// SIMATIC STEP 7 (V5.x) project ZEn01_10_STEP7__Com_SFB
// CPU: CPU414-1(1)
// CPU: CPU416-1(1)
// station: Hardware
// station: SIMATIC 400-RCV
// station: Hardware
// station: SIMATIC 400-SEND
// program: S7 Receive-Program
// program: S7 Send-Program

SYMBOL_TABLE
"IDB_USEND"	DB 8	SFB 8
"IDB_URCV"	DB 9	SFB 9
"IDB_BSEND"	DB 12	SFB 12
"IDB_BRCV"	DB 13	SFB 13
"IDB_GET"	DB 14	SFB 14
"IDB_PUT"	DB 15	SFB 15
"IDB_START"	DB 19	SFB 19
"IDB_STOP"	DB 20	SFB 20
"IDB_RESUME"	DB 21	SFB 21
"IDB_STATUS"	DB 22	SFB 22
"IDB_USTATUS"	DB 23	SFB 23
"data_usend"	DB 100	DB 100
"data_urcv"	DB 101	DB 101
"data_bsend"	DB 102	DB 102
"data_brcv"	DB 103	DB 103
"data_get"	DB 104	DB 104
"data_put"	DB 105	DB 105
"data_program_cntr"	DB 106	DB 106	// Parameters SFB START , STOP,  RESUME, STATUS and USTATUS
"data_get_source"	DB 107	DB 107
"data_put_destination"	DB 108	DB 108
"CHECK"	FC 99	FC 99	// Check the control parameters of communication function blocks
"EXAMPLE_USEND"	FC 100	FC 100
"EXAMPLE_PUT"	FC 101	FC 101
"EXAMPLE_STOP"	FC 102	FC 102
"EXAMPLE_STATUS"	FC 103	FC 103
"EXAMPLE_URCV"	FC 104	FC 104
"EXAMPLE_BSEND"	FC 105	FC 105
"EXAMPLE_BRCV"	FC 106	FC 106
"EXAMPLE_GET"	FC 107	FC 107
"EXAMPLE_START"	FC 108	FC 108
"EXAMPLE_RESUME"	FC 109	FC 109
"EXAMPLE_USTATUS"	FC 110	FC 110
"EXAMPLE_PRESET_SFBs_1"	FC 111	FC 111	// Presets on Send-CPU
"EXAMPLE_PRESET_SFBs_2"	FC 112	FC 112	// Presets on Rcv-CPU
"req_usend_user"	M 20.0	BOOL	// Trigger USEND    0->1
"req_bsend_user"	M 20.2	BOOL	// Trigger BSEND    0->1
"req_get_user"	M 20.4	BOOL	// Trigger GET    0->1
"req_put_user"	M 20.5	BOOL	// Trigger PUT   0->1
"req_start_user"	M 20.6	BOOL	// Trigger START    0->1
"req_stop_user"	M 20.7	BOOL	// Trigger STOP    0->1
"req_resume_user"	M 21.0	BOOL	// Trigger RESUME    0->1
"req_status_user"	M 21.1	BOOL	// Trigger STATUS    0->1
"req_ustatus_user"	M 21.2	BOOL	// Trigger USTATUS    0->1
"CYCL_EXC"	OB 1	OB 1	// Cycle Execution
"CYC_INT5"	OB 35	OB 35	// Cyclic Interrupt 5
"COMPLETE RESTART"	OB 100	OB 100	// Complete Restart
"USEND"	SFB 8	SFB 8	// Uncoordinated Send
"URCV"	SFB 9	SFB 9	// Uncoordinated Receive
"BSEND"	SFB 12	SFB 12	// Block Oriented Send
"BRCV"	SFB 13	SFB 13	// Block Oriented Receive
"GET"	SFB 14	SFB 14	// Read Data From a Remote CPU
"PUT"	SFB 15	SFB 15	// Write Data to a Remote CPU
"START"	SFB 19	SFB 19	// Remote Start
"STOP"	SFB 20	SFB 20	// Remote Stop
"RESUME"	SFB 21	SFB 21	// Remote Restart
"STATUS"	SFB 22	SFB 22	// Remote Status
"USTATUS"	SFB 23	SFB 23	// Receive Remote Status
"FILL"	SFC 21	SFC 21
END_SYMBOL_TABLE

FUNCTION "CHECK" : VOID	// FC 99
//This block is used to evaluate the parameters DONE/NDR/ERROR/STATUS for the 
//CFBs. 
//The parameters OK/NOT_OK are set depending on the passed parameters. 
//
VERSION : 0.0
VAR_INPUT
  ERROR : BOOL ;
  STATUS : WORD ;
  DONE_NDR : BOOL ;
END_VAR
VAR_OUTPUT
  OK : BOOL ;	// 0 Error/warning while executing CFB
  NOT_OK : BOOL ;
END_VAR
VAR_TEMP
  STAT : BOOL ;
END_VAR
BEGIN
NETWORK
TITLE = This block can be used for troubleshooting if needed
      L     #STATUS;	// Check STATUS
      L     0;
      <>I;
      =     #STAT;	// Error/warning while executing CFB 
      A     #DONE_NDR;
      =     #OK;	// CFB execution OK
      O     #STAT;	// WARNING/ERROR
      O     #ERROR;	// ERROR
      R     #OK;	// CFB execution not OK
      S     #NOT_OK;
END_FUNCTION

FUNCTION "EXAMPLE_USEND" : VOID	// FC 100
//Controlling USEND 
//
VERSION : 2.0
BEGIN
NETWORK
TITLE =
      A     "req_usend_user";	//*If "req" 0->1,
      JCN   m1;
      L     0;	//*reset 
      T     "data_usend".saved_status;	//*saved STATUS 
m1:   NOP   0;
      BLD   9;
      =     L 4.0;
      CDB;
      OPN   DI 8;
      TAR2  LD 0;
      A     "req_usend_user";
      =     DIX 0.0;
      OPN   DI 100;
      L     DIW 2;
      OPN   DI 8;
      T     DIW 2;
      OPN   DI 100;	//*If STATUS is not "0",
      L     DID 4;	//*
      OPN   DI 8;	//*
      T     DID 4;
      L     W#16#1002;	//*
      T     DIW 12;	//*set "not_ok"
      L     30;	//*and save STATUS
      T     DIW 14;
      L     100;	//*If "done"
      T     DIW 16;	//*or "error"
      L     P#DBX 10.0;	//*reset "req"
      T     DID 18;
//                                      //Add troubleshooting routine here
      L     W#16#1002;
      T     DIW 22;
      L     30;
      T     DIW 24;
      L     100;
      T     DIW 26;
      L     P#DBX 110.0;
      T     DID 28;
      L     W#16#1002;
      T     DIW 32;
      L     30;
      T     DIW 34;
      L     100;
      T     DIW 36;
      L     P#DBX 210.0;
      T     DID 38;
      L     W#16#1002;
      T     DIW 42;
      L     30;
      T     DIW 44;
      L     100;
      T     DIW 46;
      L     P#DBX 310.0;
      T     DID 48;
      LAR2  P#DBX 0.0;
      UC    "USEND";
      LAR2  LD 0;
      A     DIX 8.0;
      OPN   DI 100;
      =     DIX 0.1;
      OPN   DI 8;
      A     DIX 8.1;
      OPN   DI 100;
      =     DIX 0.2;
      OPN   DI 8;
      L     DIW 10;
      OPN   DI 100;
      T     DIW 8;
      OPN   DI 8;
      CDB;
      BLD   10;
      L     0;
      L     "data_usend".status;
      <>I;
      JCN   mark;
      SET;
      =     "data_usend".not_ok;
      T     "data_usend".saved_status;
mark: NOP   0;
      A     "data_usend".done;
      O     "data_usend".error;
      R     "req_usend_user";
      A     "data_usend".not_ok;
END_FUNCTION

FUNCTION "EXAMPLE_PUT" : VOID	// FC 101
VERSION : 2.0
BEGIN
NETWORK
TITLE =
      A     "req_put_user";	//*If "req" 0->1,
      JCN   m1;
      L     0;	//*reset 
      T     "data_put".saved_status;	//*saved STATUS 
m1:   NOP   0;
      BLD   9;
      =     L 4.0;
      CDB;
      OPN   DI 15;
      TAR2  LD 0;
      A     "req_put_user";
      =     DIX 0.0;
      OPN   DI 105;
      L     DIW 2;
      OPN   DI 15;
      T     DIW 2;
      L     W#16#1002;
      T     DIW 8;
      L     100;
      T     DIW 10;	//*If STATUS is not "0",
      L     108;	//*
      T     DIW 12;	//*
      L     P#DBX 0.0;
      T     DID 14;	//*
      L     W#16#1002;	//*set "not_ok"
      T     DIW 18;	//*and save STATUS
      L     100;
      T     DIW 20;	//*If "done"
      L     108;	//*or "error"
      T     DIW 22;	//*reset "req"
      L     P#DBX 100.0;
//                                      //Add troubleshooting routine here
      T     DID 24;
      L     W#16#1002;
      T     DIW 28;
      L     100;
      T     DIW 30;
      L     108;
      T     DIW 32;
      L     P#DBX 200.0;
      T     DID 34;
      L     W#16#1002;
      T     DIW 38;
      L     100;
      T     DIW 40;
      L     108;
      T     DIW 42;
      L     P#DBX 300.0;
      T     DID 44;
      L     W#16#1002;
      T     DIW 48;
      L     100;
      T     DIW 50;
      L     105;
      T     DIW 52;
      L     P#DBX 6.0;
      T     DID 54;
      L     W#16#1002;
      T     DIW 58;
      L     100;
      T     DIW 60;
      L     105;
      T     DIW 62;
      L     P#DBX 106.0;
      T     DID 64;
      L     W#16#1002;
      T     DIW 68;
      L     100;
      T     DIW 70;
      L     105;
      T     DIW 72;
      L     P#DBX 206.0;
      T     DID 74;
      L     W#16#1002;
      T     DIW 78;
      L     100;
      T     DIW 80;
      L     105;
      T     DIW 82;
      L     P#DBX 306.0;
      T     DID 84;
      LAR2  P#DBX 0.0;
      UC    "PUT";
      LAR2  LD 0;
      A     DIX 4.0;
      OPN   DI 105;
      =     DIX 0.1;
      OPN   DI 15;
      A     DIX 4.1;
      OPN   DI 105;
      =     DIX 0.2;
      OPN   DI 15;
      L     DIW 6;
      OPN   DI 105;
      T     DIW 4;
      OPN   DI 15;
      CDB;
      BLD   10;
      L     0;
      L     "data_put".status;
      <>I;
      JCN   mark;
      SET;
      =     "data_put".not_ok;
      T     "data_put".saved_status;
mark: NOP   0;
      A     "data_put".done;
      O     "data_put".error;
      R     "req_put_user";
      A     "data_put".not_ok;
END_FUNCTION

FUNCTION "EXAMPLE_STOP" : VOID	// FC 102
VERSION : 2.0
BEGIN
NETWORK
TITLE =
      A     "req_stop_user";	//*If "req" 0->1,
      JCN   m1;
      L     0;	//*reset 
      T     "data_program_cntr".stp_saved_status;	//*saved STATUS 
m1:   NOP   0;
      BLD   9;
      =     L 4.0;
      CDB;
      OPN   DI 20;
      TAR2  LD 0;
      A     "req_stop_user";
      =     DIX 0.0;
      OPN   DI 106;
      L     DIW 18;	//*If STATUS is not "0",
      OPN   DI 20;	//*
      T     DIW 2;	//*
      L     W#16#1002;
      T     DIW 8;	//*
      L     10;	//*set "not_ok"
      T     DIW 10;	//*and save STATUS
      L     106;
      T     DIW 12;	//*If "done"
      L     P#DBX 0.0;	//*or "error"
      T     DID 14;	//*reset "req"
      OPN   DI 106;	//                                      //Add troubleshooting routine here
      L     DIB 22;
      OPN   DI 20;
      T     DIB 18;
      LAR2  P#DBX 0.0;
      UC    "STOP";
      LAR2  LD 0;
      A     DIX 4.0;
      OPN   DI 106;
      =     DIX 17.1;
      OPN   DI 20;
      A     DIX 4.1;
      OPN   DI 106;
      =     DIX 17.2;
      OPN   DI 20;
      L     DIW 6;
      OPN   DI 106;
      T     DIW 20;
      OPN   DI 20;
      L     DIB 18;
      OPN   DI 106;
      T     DIB 22;
      OPN   DI 20;
      CDB;
      BLD   10;
      L     0;
      L     "data_program_cntr".stop_status;
      <>I;
      JCN   mark;
      SET;
      =     "data_program_cntr".stop_not_ok;
      T     "data_program_cntr".stp_saved_status;
mark: NOP   0;
      A     "data_program_cntr".stop_done;
      O     "data_program_cntr".stop_error;
      R     "req_stop_user";
      A     "data_program_cntr".stop_not_ok;
END_FUNCTION

FUNCTION "EXAMPLE_STATUS" : VOID	// FC 103
VERSION : 2.0
BEGIN
NETWORK
TITLE =
      A     "req_status_user";	//*If "req" 0->1,
      JCN   m1;
      L     0;	//*reset 
      T     "data_program_cntr".sta_saved_status;	//*saved STATUS 
m1:   NOP   0;
      BLD   9;
      =     L 4.0;
      CDB;
      OPN   DI 22;
      TAR2  LD 0;
      A     "req_status_user";
      =     DIX 0.0;
      OPN   DI 106;
      L     DIW 30;
      OPN   DI 22;	//*If STATUS is not "0",
      T     DIW 2;	//*
      L     W#16#1004;	//*
      T     DIW 8;
      L     1;	//*
      T     DIW 10;	//*set "not_ok"
      L     106;	//*and save STATUS
      T     DIW 12;
      L     P#DBX 34.0;	//*If "done"
      T     DID 14;	//*or "error"
      L     W#16#1004;	//*reset "req"
      T     DIW 18;
//                                      //Add troubleshooting routine here
      L     1;
      T     DIW 20;
      L     106;
      T     DIW 22;
      L     P#DBX 36.0;
      T     DID 24;
      L     W#16#1004;
      T     DIW 28;
      L     1;
      T     DIW 30;
      L     106;
      T     DIW 32;
      L     P#DBX 38.0;
      T     DID 34;
      LAR2  P#DBX 0.0;
      UC    "STATUS";
      LAR2  LD 0;
      A     DIX 4.0;
      OPN   DI 106;
      =     DIX 29.1;
      OPN   DI 22;
      A     DIX 4.1;
      OPN   DI 106;
      =     DIX 29.2;
      OPN   DI 22;
      L     DIW 6;
      OPN   DI 106;
      T     DIW 32;
      OPN   DI 22;
      CDB;
      BLD   10;
      L     0;
      L     "data_program_cntr".status_status;
      <>I;
      JCN   mark;
      SET;
      =     "data_program_cntr".status_not_ok;
      T     "data_program_cntr".sta_saved_status;
mark: NOP   0;
      A     "data_program_cntr".status_done;
      O     "data_program_cntr".status_error;
      R     "req_status_user";
      A     "data_program_cntr".status_not_ok;
END_FUNCTION

FUNCTION "EXAMPLE_BSEND" : VOID	// FC 105
//Controlling BSEND 
//
VERSION : 2.0
BEGIN
NETWORK
TITLE =
      A     "req_bsend_user";	//*If "req" 0->1,
      JCN   m1;
      L     0;	//*reset 
      T     "data_bsend".saved_status;	//*saved STATUS 
m1:   NOP   0;
      BLD   9;
      =     L 4.0;
      CDB;
      OPN   DI 12;
      TAR2  LD 0;
      A     "req_bsend_user";
      =     DIX 0.0;
      OPN   DI 102;
      L     DIW 2;
      OPN   DI 12;
      T     DIW 2;	//*If STATUS is not "0",
      OPN   DI 102;	//*
      L     DID 4;	//*
      OPN   DI 12;
      T     DID 4;	//*
      L     W#16#1002;	//*set "not_ok"
      T     DIW 12;	//*and save STATUS
      L     500;
      T     DIW 14;	//*If "done"
      L     102;	//*or "error"
      T     DIW 16;	//*reset "req"
      L     P#DBX 12.0;
//                                      //Add troubleshooting routine here
      T     DID 18;
      OPN   DI 102;
      L     DIW 10;
      OPN   DI 12;
      T     DIW 22;
      LAR2  P#DBX 0.0;
      UC    "BSEND";
      LAR2  LD 0;
      A     DIX 8.0;
      OPN   DI 102;
      =     DIX 0.1;
      OPN   DI 12;
      A     DIX 8.1;
      OPN   DI 102;
      =     DIX 0.2;
      OPN   DI 12;
      L     DIW 10;
      OPN   DI 102;
      T     DIW 8;
      OPN   DI 12;
      L     DIW 22;
      OPN   DI 102;
      T     DIW 10;
      OPN   DI 12;
      CDB;
      BLD   10;
      L     0;
      L     "data_bsend".status;
      <>I;
      JCN   mark;
      SET;
      =     "data_bsend".not_ok;
      T     "data_bsend".saved_status;
mark: NOP   0;
      A     "data_bsend".done;
      O     "data_bsend".error;
      R     "req_bsend_user";
      A     "data_bsend".not_ok;
END_FUNCTION

FUNCTION "EXAMPLE_GET" : VOID	// FC 107
VERSION : 2.0
BEGIN
NETWORK
TITLE =
      A     "req_get_user";	//*If "req" 0->1,
      JCN   m1;
      L     0;	//*reset 
      T     "data_get".saved_status;	//*saved STATUS 
m1:   NOP   0;
      BLD   9;
      =     L 4.0;
      CDB;
      OPN   DI 14;
      TAR2  LD 0;
      A     "req_get_user";
      =     DIX 0.0;
      OPN   DI 104;
      L     DIW 2;
      OPN   DI 14;
      T     DIW 2;
      L     W#16#1002;
      T     DIW 8;
      L     100;
      T     DIW 10;	//*If STATUS is not "0",
      L     107;	//*
      T     DIW 12;	//*
      L     P#DBX 0.0;
      T     DID 14;	//*
      L     W#16#1002;	//*set "not_ok"
      T     DIW 18;	//*and save STATUS
      L     100;
      T     DIW 20;	//*If "done"
      L     107;	//*or "error"
      T     DIW 22;	//*reset "req"
      L     P#DBX 100.0;
//                                      //Add troubleshooting routine here
      T     DID 24;
      L     W#16#1002;
      T     DIW 28;
      L     100;
      T     DIW 30;
      L     107;
      T     DIW 32;
      L     P#DBX 200.0;
      T     DID 34;
      L     W#16#1002;
      T     DIW 38;
      L     100;
      T     DIW 40;
      L     107;
      T     DIW 42;
      L     P#DBX 300.0;
      T     DID 44;
      L     W#16#1002;
      T     DIW 48;
      L     100;
      T     DIW 50;
      L     104;
      T     DIW 52;
      L     P#DBX 6.0;
      T     DID 54;
      L     W#16#1002;
      T     DIW 58;
      L     100;
      T     DIW 60;
      L     104;
      T     DIW 62;
      L     P#DBX 106.0;
      T     DID 64;
      L     W#16#1002;
      T     DIW 68;
      L     100;
      T     DIW 70;
      L     104;
      T     DIW 72;
      L     P#DBX 206.0;
      T     DID 74;
      L     W#16#1002;
      T     DIW 78;
      L     100;
      T     DIW 80;
      L     104;
      T     DIW 82;
      L     P#DBX 306.0;
      T     DID 84;
      LAR2  P#DBX 0.0;
      UC    "GET";
      LAR2  LD 0;
      A     DIX 4.0;
      OPN   DI 104;
      =     DIX 0.1;
      OPN   DI 14;
      A     DIX 4.1;
      OPN   DI 104;
      =     DIX 0.2;
      OPN   DI 14;
      L     DIW 6;
      OPN   DI 104;
      T     DIW 4;
      OPN   DI 14;
      CDB;
      BLD   10;
      L     0;
      L     "data_get".status;
      <>I;
      JCN   mark;
      SET;
      =     "data_get".not_ok;
      T     "data_get".saved_status;
mark: NOP   0;
      A     "data_get".ndr;
      O     "data_get".error;
      R     "req_get_user";
      A     "data_get".not_ok;
END_FUNCTION

FUNCTION "EXAMPLE_START" : VOID	// FC 108
VERSION : 2.0
BEGIN
NETWORK
TITLE =
      A     "req_start_user";	//*If "req" 0->1,
      JCN   m1;
      L     0;	//*reset 
      T     "data_program_cntr".stt_saved_status;	//*saved STATUS 
m1:   NOP   0;
      BLD   9;
      =     L 4.0;
      CDB;
      OPN   DI 19;
      TAR2  LD 0;
      A     "req_start_user";
      =     DIX 0.0;
      OPN   DI 106;
      L     DIW 12;
      OPN   DI 19;	//*If STATUS is not "0",
      T     DIW 2;	//*
      L     W#16#1002;	//*
      T     DIW 8;
      L     10;	//*
      T     DIW 10;	//*set "not_ok"
      L     106;	//*and save STATUS
      T     DIW 12;
      L     P#DBX 0.0;	//*If "done"
      T     DID 14;	//*or "error"
      OPN   DI 106;	//*reset "req"
      L     DIB 16;
//                                      //Add troubleshooting routine here
      OPN   DI 19;
      T     DIB 28;
      LAR2  P#DBX 0.0;
      UC    "START";
      LAR2  LD 0;
      A     DIX 4.0;
      OPN   DI 106;
      =     DIX 10.1;
      OPN   DI 19;
      A     DIX 4.1;
      OPN   DI 106;
      =     DIX 10.2;
      OPN   DI 19;
      L     DIW 6;
      OPN   DI 106;
      T     DIW 14;
      OPN   DI 19;
      L     DIB 28;
      OPN   DI 106;
      T     DIB 16;
      OPN   DI 19;
      CDB;
      BLD   10;
      L     0;
      L     "data_program_cntr".start_status;
      <>I;
      JCN   mark;
      SET;
      =     "data_program_cntr".start_not_ok;
      T     "data_program_cntr".stt_saved_status;
mark: NOP   0;
      A     "data_program_cntr".start_done;
      O     "data_program_cntr".start_error;
      R     "req_start_user";
      A     "data_program_cntr".start_not_ok;
END_FUNCTION

FUNCTION "EXAMPLE_RESUME" : VOID	// FC 109
//To use this block, you have to activate "Warmrestart"in HARDWARE-Configuration
//and on the CPU you have to set the "CRST/WRST -switch" into WRST-Mode
VERSION : 2.0
BEGIN
NETWORK
TITLE =
      A     "req_resume_user";	//*If "req" 0->1,
      JCN   m1;
      L     0;	//*reset 
      T     "data_program_cntr".res_saved_status;	//*saved STATUS 
m1:   NOP   0;
      BLD   9;
      =     L 4.0;
      CDB;
      OPN   DI 21;
      TAR2  LD 0;
      A     "req_resume_user";
      =     DIX 0.0;
      OPN   DI 106;
      L     DIW 24;
      OPN   DI 21;	//*If STATUS is not "0",
      T     DIW 2;	//*
      L     W#16#1002;	//*
      T     DIW 8;
      L     10;	//*
      T     DIW 10;	//*set "not_ok"
      L     106;	//*and save STATUS
      T     DIW 12;
      L     P#DBX 0.0;	//*If "done"
      T     DID 14;	//*or "error"
      OPN   DI 106;	//*reset "req"
      L     DIB 28;
//                                      //Add troubleshooting routine here
      OPN   DI 21;
      T     DIB 28;
      LAR2  P#DBX 0.0;
      UC    "RESUME";
      LAR2  LD 0;
      A     DIX 4.0;
      OPN   DI 106;
      =     DIX 23.1;
      OPN   DI 21;
      A     DIX 4.1;
      OPN   DI 106;
      =     DIX 23.2;
      OPN   DI 21;
      L     DIW 6;
      OPN   DI 106;
      T     DIW 26;
      OPN   DI 21;
      L     DIB 28;
      OPN   DI 106;
      T     DIB 28;
      OPN   DI 21;
      CDB;
      BLD   10;
      L     0;
      L     "data_program_cntr".resume_status;
      <>I;
      JCN   mark;
      SET;
      =     "data_program_cntr".resume_not_ok;
      T     "data_program_cntr".res_saved_status;
mark: NOP   0;
      A     "data_program_cntr".resume_done;
      O     "data_program_cntr".resume_error;
      R     "req_resume_user";
      A     "data_program_cntr".resume_not_ok;
END_FUNCTION

FUNCTION "EXAMPLE_USTATUS" : VOID	// FC 110
//You can only use this block, if in CONNECTION TABLE you have activated "SEND 
//OPERATING MODE MESSAGES"!! 
//
VERSION : 0.0
BEGIN
NETWORK
TITLE =
      A     "req_ustatus_user";	//*If "en_r" 0->1,
      FP    "data_program_cntr".edge_usta;
      JCN   m1;
      L     0;	//*reset 
      T     "data_program_cntr".usta_saved_status;	//*saved STATUS 
m1:   NOP   0;
      BLD   9;
      =     L 4.0;
      CDB;
      OPN   DI 23;
      TAR2  LD 0;
      A     "req_ustatus_user";
      =     DIX 0.0;
      OPN   DI 106;
      L     DIW 42;
      OPN   DI 23;	//*If STATUS is not "0",
      T     DIW 2;	//*
      L     W#16#1004;	//*
      T     DIW 8;
      L     1;	//*
      T     DIW 10;	//*set "not_ok"
      L     106;	//*and save STATUS
      T     DIW 12;
      L     P#DBX 46.0;
//                                      //Add troubleshooting routine here
      T     DID 14;
      L     W#16#1004;
      T     DIW 18;
      L     1;
      T     DIW 20;
      L     106;
      T     DIW 22;
      L     P#DBX 48.0;
      T     DID 24;
      L     W#16#1004;
      T     DIW 28;
      L     1;
      T     DIW 30;
      L     106;
      T     DIW 32;
      L     P#DBX 50.0;
      T     DID 34;
      LAR2  P#DBX 0.0;
      UC    "USTATUS";
      LAR2  LD 0;
      A     DIX 4.0;
      OPN   DI 106;
      =     DIX 40.1;
      OPN   DI 23;
      A     DIX 4.1;
      OPN   DI 106;
      =     DIX 40.2;
      OPN   DI 23;
      L     DIW 6;
      OPN   DI 106;
      T     DIW 44;
      OPN   DI 23;
      CDB;
      BLD   10;
      L     0;
      L     "data_program_cntr".ustatus_status;
      <>I;
      JCN   mark;
      SET;
      =     "data_program_cntr".ustatus_not_ok;
      T     "data_program_cntr".usta_saved_status;
mark: NOP   0;
      A     "data_program_cntr".ustatus_not_ok;
END_FUNCTION

FUNCTION "EXAMPLE_PRESET_SFBs_1" : VOID	// FC 111
TITLE = *****              INITIALIZING CFBs           *****
VERSION : 2.0
BEGIN
NETWORK
TITLE =   Defining the PI_NAME 
//for SIMATIC S7-Systems PI_NAME = P_PROGRAM
      L     'P_';
      T     "data_program_cntr".pi_name[1];
      L     'PR';
      T     "data_program_cntr".pi_name[2];
      L     'OG';
      T     "data_program_cntr".pi_name[3];
      L     'RA';
      T     "data_program_cntr".pi_name[4];
      L     'M ';
      T     "data_program_cntr".pi_name[5];
//*******************************************************
NETWORK
TITLE =  INITIALIZING USEND 
      CLR;
      =     "req_usend_user";
      L     W#16#1;	// connection_id
      T     "data_usend".id;
      L     DW#16#80009;
      T     "data_usend".r_id;
      L     W#16#0;	//Reset saved STATUS
      T     "data_usend".saved_status;
NETWORK
TITLE =  INITIALIZING BSEND 
      CLR;
      =     "req_bsend_user";
      L     W#16#1;	// connection_id
      T     "data_bsend".id;
      L     DW#16#C000D;
      T     "data_bsend".r_id;
      L     W#16#1F4;
      T     "data_bsend".len;
      L     W#16#0;	//Reset saved STATUS
      T     "data_bsend".saved_status;
NETWORK
TITLE =  INITIALIZING GET 
      CLR;
      =     "req_get_user";
      L     W#16#1;	// connection_id
      T     "data_get".id;
      L     W#16#0;	//Reset saved STATUS
      T     "data_get".saved_status;
NETWORK
TITLE =  INITIALIZING PUT 
      CLR;
      =     "req_put_user";
      L     W#16#1;	// connection_id
      T     "data_put".id;
      L     W#16#0;	//Reset saved STATUS
      T     "data_put".saved_status;
NETWORK
TITLE =   INITIALIZING START 
      CLR;
      =     "req_start_user";
      L     W#16#1;	// connection_id
      T     "data_program_cntr".start_id;
      L     W#16#0;	//Reset saved STATUS
      T     "data_program_cntr".stt_saved_status;
NETWORK
TITLE =   INITIALIZING STOP 
      CLR;
      =     "req_stop_user";
      L     W#16#1;	// connection_id
      T     "data_program_cntr".stop_id;
      L     W#16#0;	//Reset saved STATUS
      T     "data_program_cntr".stp_saved_status;
NETWORK
TITLE =   INITIALIZING RESUME 
      CLR;
      =     "req_resume_user";
      L     W#16#1;	// connection_id
      T     "data_program_cntr".resume_id;
      L     W#16#0;	//Reset saved STATUS
      T     "data_program_cntr".res_saved_status;
NETWORK
TITLE =  INITIALIZING STATUS               
      CLR;
      =     "req_status_user";
      L     W#16#1;	// connection_id
      T     "data_program_cntr".status_id;
      L     W#16#0;	//Reset saved STATUS
      T     "data_program_cntr".sta_saved_status;
NETWORK
TITLE =  INITIALIZING USTATUS                 
      CLR;
      =     "req_ustatus_user";
      L     W#16#1;	// connection_id
      T     "data_program_cntr".ustatus_id;
      L     W#16#0;	//Reset saved STATUS
      T     "data_program_cntr".usta_saved_status;
NETWORK
TITLE =  Presetting the send values for USEND 
// Data_usend.send_data_1..4
//
      L     W#16#101;
      T     "data_usend".fill_1;
      CALL  "FILL" (
           BVAL                     := "data_usend".fill_1,
           RET_VAL                  := "data_usend".ret_val,
           BLK                      := "data_usend".send_data_1);
      L     W#16#202;
      T     "data_usend".fill_2;
      CALL  "FILL" (
           BVAL                     := "data_usend".fill_2,
           RET_VAL                  := "data_usend".ret_val,
           BLK                      := "data_usend".send_data_2);
      L     W#16#303;
      T     "data_usend".fill_3;
      CALL  "FILL" (
           BVAL                     := "data_usend".fill_3,
           RET_VAL                  := "data_usend".ret_val,
           BLK                      := "data_usend".send_data_3);
      L     W#16#404;
      T     "data_usend".fill_4;
      CALL  "FILL" (
           BVAL                     := "data_usend".fill_4,
           RET_VAL                  := "data_usend".ret_val,
           BLK                      := "data_usend".send_data_4);
NETWORK
TITLE = Presetting send data SFB BSEND
//send data length = 1000 byte
      L     W#16#101;
      T     "data_bsend".fill_1;
      CALL  "FILL" (
           BVAL                     := "data_bsend".fill_1,
           RET_VAL                  := "data_bsend".ret_val,
           BLK                      := "data_bsend".send_data_1);
NETWORK
TITLE = Reset Data Area SFB GET 
//rcv data = 4 x 100 byte filled with b#16#00
//
      L     B#16#0;
      T     "data_get".fill;
      CALL  "FILL" (
           BVAL                     := "data_get".fill,
           RET_VAL                  := "data_get".ret_val,
           BLK                      := "data_get".rcv_data_1);
      CALL  "FILL" (
           BVAL                     := "data_get".fill,
           RET_VAL                  := "data_get".ret_val,
           BLK                      := "data_get".rcv_data_2);
      CALL  "FILL" (
           BVAL                     := "data_get".fill,
           RET_VAL                  := "data_get".ret_val,
           BLK                      := "data_get".rcv_data_3);
      CALL  "FILL" (
           BVAL                     := "data_get".fill,
           RET_VAL                  := "data_get".ret_val,
           BLK                      := "data_get".rcv_data_4);
NETWORK
TITLE = Presetting SEND data SFB PUT
//send data = 4 x 100 byte
//
      L     W#16#1111;
      T     "data_put".fill_1;
      CALL  "FILL" (
           BVAL                     := "data_put".fill_1,
           RET_VAL                  := "data_put".ret_val,
           BLK                      := "data_put".send_data_1);
      L     W#16#2222;
      T     "data_put".fill_2;
      CALL  "FILL" (
           BVAL                     := "data_put".fill_2,
           RET_VAL                  := "data_put".ret_val,
           BLK                      := "data_put".send_data_2);
      L     W#16#3333;
      T     "data_put".fill_3;
      CALL  "FILL" (
           BVAL                     := "data_put".fill_3,
           RET_VAL                  := "data_put".ret_val,
           BLK                      := "data_put".send_data_3);
      L     W#16#4444;
      T     "data_put".fill_4;
      CALL  "FILL" (
           BVAL                     := "data_put".fill_4,
           RET_VAL                  := "data_put".ret_val,
           BLK                      := "data_put".send_data_4);
NETWORK
TITLE = BLOCK_END
END_FUNCTION

DATA_BLOCK "IDB_USEND"	// DB 8
VERSION : 0.0
"USEND"
BEGIN
END_DATA_BLOCK

DATA_BLOCK "IDB_BSEND"	// DB 12
VERSION : 0.0
"BSEND"
BEGIN
END_DATA_BLOCK

DATA_BLOCK "IDB_GET"	// DB 14
VERSION : 0.0
"GET"
BEGIN
END_DATA_BLOCK

DATA_BLOCK "IDB_PUT"	// DB 15
VERSION : 0.0
"PUT"
BEGIN
END_DATA_BLOCK

DATA_BLOCK "IDB_START"	// DB 19
VERSION : 0.0
"START"
BEGIN
END_DATA_BLOCK

DATA_BLOCK "IDB_STOP"	// DB 20
VERSION : 0.0
"STOP"
BEGIN
END_DATA_BLOCK

DATA_BLOCK "IDB_RESUME"	// DB 21
VERSION : 0.0
"RESUME"
BEGIN
END_DATA_BLOCK

DATA_BLOCK "IDB_STATUS"	// DB 22
VERSION : 0.0
"STATUS"
BEGIN
END_DATA_BLOCK

DATA_BLOCK "IDB_USTATUS"	// DB 23
VERSION : 0.0
"USTATUS"
BEGIN
END_DATA_BLOCK

DATA_BLOCK "data_usend"	// DB 100
VERSION : 0.0
  STRUCT
   req : BOOL ;	//Can be used if needed
   done : BOOL ;
   error : BOOL ;
   busy : BOOL ;	//Can be used if needed
   ok : BOOL ;
   not_ok : BOOL ;
   id : WORD ;
   r_id : DWORD ;
   status : WORD ;
   send_data_1 : ARRAY  [1 .. 30 ] OF BYTE ;
   dummy_1 : ARRAY  [1 .. 70 ] OF BYTE ;
   send_data_2 : ARRAY  [1 .. 30 ] OF BYTE ;
   dummy_2 : ARRAY  [1 .. 70 ] OF BYTE ;
   send_data_3 : ARRAY  [1 .. 30 ] OF BYTE ;
   dummy_3 : ARRAY  [1 .. 70 ] OF BYTE ;
   send_data_4 : ARRAY  [1 .. 30 ] OF BYTE ;
   dummy_4 : ARRAY  [1 .. 70 ] OF BYTE ;
   fill_1 : WORD ;
   fill_2 : WORD ;
   fill_3 : WORD ;
   fill_4 : WORD ;
   ret_val : INT ;
   saved_status : WORD ;
  END_STRUCT ;	
BEGIN
END_DATA_BLOCK

DATA_BLOCK "data_bsend"	// DB 102
VERSION : 0.0
  STRUCT
   req : BOOL ;	//Can be used if needed
   done : BOOL ;
   error : BOOL ;
   busy : BOOL ;	//Can be used if needed
   ok : BOOL ;
   not_ok : BOOL ;
   id : WORD ;
   r_id : DWORD ;
   status : WORD ;
   len : WORD ;
   send_data_1 : ARRAY  [1 .. 500 ] OF BYTE ;
   dummy_1 : ARRAY  [1 .. 500 ] OF BYTE ;
   fill_1 : WORD ;
   ret_val : INT ;
   saved_status : WORD ;
  END_STRUCT ;	
BEGIN
END_DATA_BLOCK

DATA_BLOCK "data_get"	// DB 104
VERSION : 0.0
  STRUCT
   req : BOOL ;	//Can be used if needed
   ndr : BOOL ;
   error : BOOL ;
   busy : BOOL ;	//Can be used if needed
   ok : BOOL ;
   not_ok : BOOL ;
   id : WORD ;
   status : WORD ;
   rcv_data_1 : ARRAY  [1 .. 100 ] OF BYTE ;
   rcv_data_2 : ARRAY  [1 .. 100 ] OF BYTE ;
   rcv_data_3 : ARRAY  [1 .. 100 ] OF BYTE ;
   rcv_data_4 : ARRAY  [1 .. 100 ] OF BYTE ;
   fill : WORD ;
   ret_val : INT ;	//ret_val des sfc FILL
   saved_status : WORD ;
  END_STRUCT ;	
BEGIN
   error := TRUE;
   id := W#16#1;
   status := W#16#4;
END_DATA_BLOCK

DATA_BLOCK "data_put"	// DB 105
VERSION : 0.0
  STRUCT
   req : BOOL ;	//Can be used if needed
   done : BOOL ;
   error : BOOL ;
   busy : BOOL ;	//Can be used if needed
   ok : BOOL ;
   not_ok : BOOL ;
   id : WORD ;
   status : WORD ;
   send_data_1 : ARRAY  [1 .. 100 ] OF BYTE ;
   send_data_2 : ARRAY  [1 .. 100 ] OF BYTE ;
   send_data_3 : ARRAY  [1 .. 100 ] OF BYTE ;
   send_data_4 : ARRAY  [1 .. 100 ] OF BYTE ;
   fill_1 : WORD ;
   fill_2 : WORD ;
   fill_3 : WORD ;
   fill_4 : WORD ;
   ret_val : INT ;
   saved_status : WORD ;
  END_STRUCT ;	
BEGIN
END_DATA_BLOCK

DATA_BLOCK "data_program_cntr"	// DB 106
VERSION : 2.0
  STRUCT
   pi_name : ARRAY  [1 .. 5 ] OF WORD ;
   start_req : BOOL ;	//Can be used if needed
   start_done : BOOL ;
   start_error : BOOL ;
   start_busy : BOOL ;	//Can be used if needed
   start_ok : BOOL ;
   start_not_ok : BOOL ;
   start_id : WORD ;
   start_status : WORD ;
   start_io_state : BYTE ;
   stop_req : BOOL ;	//Can be used if needed
   stop_done : BOOL ;
   stop_error : BOOL ;
   stop_busy : BOOL ;	//Can be used if needed
   stop_ok : BOOL ;
   stop_not_ok : BOOL ;
   stop_id : WORD ;
   stop_status : WORD ;
   stop_io_state : BYTE ;
   resume_req : BOOL ;	//Can be used if needed
   resume_done : BOOL ;
   resume_error : BOOL ;
   resume_busy : BOOL ;	//Can be used if needed
   resume_ok : BOOL ;
   resume_not_ok : BOOL ;
   resume_id : WORD ;
   resume_status : WORD ;
   resume_io_state : BYTE ;
   status_req : BOOL ;	//Can be used if needed
   status_done : BOOL ;
   status_error : BOOL ;
   status_busy : BOOL ;	//Can be used if needed
   status_ok : BOOL ;
   status_not_ok : BOOL ;
   status_id : WORD ;
   status_status : WORD ;
   status_phys : WORD ;
   status_loc : WORD ;
   status_local : WORD ;
   ustatus_en_r : BOOL ;	//Can be used if needed
   ustatus_ndr : BOOL ;
   ustatus_error : BOOL ;
   ustatus_busy : BOOL ;	//Can be used if needed
   ustatus_ok : BOOL ;
   ustatus_not_ok : BOOL ;
   ustatus_id : WORD ;
   ustatus_status : WORD ;
   ustatus_phys : WORD ;
   ustatus_loc : WORD ;
   ustatus_local : WORD ;
   stt_saved_status : WORD ;
   stp_saved_status : WORD ;
   res_saved_status : WORD ;
   sta_saved_status : WORD ;
   usta_saved_status : WORD ;
   edge_usta : BOOL ;
  END_STRUCT ;	
BEGIN
END_DATA_BLOCK

DATA_BLOCK "data_get_source"	// DB 107
VERSION : 0.1
  STRUCT
   source_1 : ARRAY  [1 .. 100 ] OF BYTE ;
   source_2 : ARRAY  [1 .. 100 ] OF BYTE ;
   source_3 : ARRAY  [1 .. 100 ] OF BYTE ;
   source_4 : ARRAY  [1 .. 100 ] OF BYTE ;
  END_STRUCT ;	
BEGIN
END_DATA_BLOCK

DATA_BLOCK "data_put_destination"	// DB 108
VERSION : 0.1
  STRUCT
   dest_1 : ARRAY  [1 .. 100 ] OF BYTE ;
   dest_2 : ARRAY  [1 .. 100 ] OF BYTE ;
   dest_3 : ARRAY  [1 .. 100 ] OF BYTE ;
   dest_4 : ARRAY  [1 .. 100 ] OF BYTE ;
  END_STRUCT ;	
BEGIN
END_DATA_BLOCK

ORGANIZATION_BLOCK "CYCL_EXC"	// OB 1
VERSION : 0.1
VAR_TEMP
  OB1_EV_CLASS : BYTE ;	//Bits 0-3 = 1 (Coming event), Bits 4-7 = 1 (Event class 1)
  OB1_SCAN_1 : BYTE ;	//1 (Cold restart scan 1 of OB 1), 3 (Scan 2-n of OB 1)
  OB1_PRIORITY : BYTE ;	//1 (Priority of 1 is lowest)
  OB1_OB_NUMBR : BYTE ;	//1 (Organization block 1, OB1)
  OB1_RESERVED_1 : BYTE ;	//Reserved for system
  OB1_RESERVED_2 : BYTE ;	//Reserved for system
  OB1_PREV_CYCLE : INT ;	//Cycle time of previous OB1 scan (milliseconds)
  OB1_MIN_CYCLE : INT ;	//Minimum cycle time of OB1 (milliseconds)
  OB1_MAX_CYCLE : INT ;	//Maximum cycle time of OB1 (milliseconds)
  OB1_DATE_TIME : DATE_AND_TIME ;	//Date and time OB1 started
END_VAR
BEGIN
NETWORK
TITLE =
END_ORGANIZATION_BLOCK

ORGANIZATION_BLOCK "CYC_INT5"	// OB 35
TITLE = "100 ms Cycle"
VERSION : 1.0
VAR_TEMP
  OB35_EV_CLASS : BYTE ;
  OB35_STRT_INF : BYTE ;
  OB35_PRIORITY : BYTE ;
  OB35_OB_NUMBR : BYTE ;
  OB35_RESERVED_1 : BYTE ;
  OB35_RESERVED_2 : BYTE ;
  OB35_PHASE_OFFSET : WORD ;
  OB35_RESERVED_3 : INT ;
  OB35_EXC_FREQ : INT ;
  OB35_DATE_TIME : DATE_AND_TIME ;
END_VAR
BEGIN
NETWORK
TITLE =   CALL USEND 
      CALL  "EXAMPLE_USEND";
NETWORK
TITLE =  CALL BSEND 
      CALL  "EXAMPLE_BSEND";
NETWORK
TITLE =   CALL  GET
      CALL  "EXAMPLE_GET";
NETWORK
TITLE =   CALL   PUT
      CALL  "EXAMPLE_PUT";
NETWORK
TITLE =  CALL START 
      CALL  "EXAMPLE_START";
NETWORK
TITLE =   CALL  STOP
      CALL  "EXAMPLE_STOP";
NETWORK
TITLE =   CALL  RESUME 
      CALL  "EXAMPLE_RESUME";
NETWORK
TITLE =   CALL  STATUS
      CALL  "EXAMPLE_STATUS";
NETWORK
TITLE =  CALL USTATUS
      CALL  "EXAMPLE_USTATUS";
END_ORGANIZATION_BLOCK

ORGANIZATION_BLOCK "COMPLETE RESTART"	// OB 100
TITLE = "Complete Restart"
VERSION : 1.0
VAR_TEMP
  OB100_EV_CLASS : BYTE ;
  OB100_STRTUP : BYTE ;
  OB100_PRIORITY : BYTE ;
  OB100_OB_NUMBR : BYTE ;
  OB100_RESERVED_1 : BYTE ;
  OB100_RESERVED_2 : BYTE ;
  OB100_STOP : WORD ;
  OB100_STRT_INFO : DWORD ;
  OB100_DATE_TIME : DATE_AND_TIME ;
END_VAR
BEGIN
NETWORK
TITLE =
      CALL  "EXAMPLE_PRESET_SFBs_1";
END_ORGANIZATION_BLOCK

SYMBOL_TABLE
"IDB_USEND"	DB 8	SFB 8
"IDB_URCV"	DB 9	SFB 9
"IDB_BSEND"	DB 12	SFB 12
"IDB_BRCV"	DB 13	SFB 13
"IDB_GET"	DB 14	SFB 14
"IDB_PUT"	DB 15	SFB 15
"IDB_START"	DB 19	SFB 19
"IDB_STOP"	DB 20	SFB 20
"IDB_RESUME"	DB 21	SFB 21
"IDB_STATUS"	DB 22	SFB 22
"IDB_USTATUS"	DB 23	SFB 23
"data_usend"	DB 100	DB 100
"data_urcv"	DB 101	DB 101
"data_bsend"	DB 102	DB 102
"data_brcv"	DB 103	DB 103
"data_get"	DB 104	DB 104
"data_put"	DB 105	DB 105
"data_program_cntr"	DB 106	DB 106	// Parameters SFB START , STOP,  RESUME, STATUS and USTATUS
"data_get_source"	DB 107	DB 107
"data_put_destination"	DB 108	DB 108
"CHECK"	FC 99	FC 99	// Check the control parameters of communication function blocks
"EXAMPLE_USEND"	FC 100	FC 100
"EXAMPLE_PUT"	FC 101	FC 101
"EXAMPLE_STOP"	FC 102	FC 102
"EXAMPLE_STATUS"	FC 103	FC 103
"EXAMPLE_URCV"	FC 104	FC 104
"EXAMPLE_BSEND"	FC 105	FC 105
"EXAMPLE_BRCV"	FC 106	FC 106
"EXAMPLE_GET"	FC 107	FC 107
"EXAMPLE_START"	FC 108	FC 108
"EXAMPLE_RESUME"	FC 109	FC 109
"EXAMPLE_USTATUS"	FC 110	FC 110
"EXAMPLE_PRESET_SFBs_1"	FC 111	FC 111	// Presets on Send-CPU
"EXAMPLE_PRESET_SFBs_2"	FC 112	FC 112	// Presets on Rcv-CPU
"en_r_urcv_user"	M 20.1	BOOL	// Start URCV    =1
"en_r_brcv_user"	M 20.3	BOOL	// Start BRCV    =1
"CYCL_EXC"	OB 1	OB 1	// Cycle Execution
"CYC_INT5"	OB 35	OB 35	// Cyclic Interrupt 5
"COMPLETE RESTART"	OB 100	OB 100	// Complete Restart
"USEND"	SFB 8	SFB 8	// Uncoordinated Send
"URCV"	SFB 9	SFB 9	// Uncoordinated Receive
"BSEND"	SFB 12	SFB 12	// Block Oriented Send
"BRCV"	SFB 13	SFB 13	// Block Oriented Receive
"GET"	SFB 14	SFB 14	// Read Data From a Remote CPU
"PUT"	SFB 15	SFB 15	// Write Data to a Remote CPU
"START"	SFB 19	SFB 19	// Remote Start
"STOP"	SFB 20	SFB 20	// Remote Stop
"RESUME"	SFB 21	SFB 21	// Remote Restart
"STATUS"	SFB 22	SFB 22	// Remote Status
"USTATUS"	SFB 23	SFB 23	// Receive Remote Status
"FILL"	SFC 21	SFC 21
END_SYMBOL_TABLE

FUNCTION "CHECK" : VOID	// FC 99
//This block is used to evaluate the parameters DONE/NDR/ERROR/STATUS for the 
//CFBs. 
//The parameters OK/NOT_OK are set depending on the passed parameters. 
//
VERSION : 0.0
VAR_INPUT
  ERROR : BOOL ;
  STATUS : WORD ;
  DONE_NDR : BOOL ;
END_VAR
VAR_OUTPUT
  OK : BOOL ;	// 0 Error/warning while executing CFB
  NOT_OK : BOOL ;
END_VAR
VAR_TEMP
  STAT : BOOL ;
END_VAR
BEGIN
NETWORK
TITLE = This block can be used for troubleshooting if needed
      L     #STATUS;	// Check STATUS
      L     0;
      <>I;
      =     #STAT;	// Error/warning while executing CFB 
      A     #DONE_NDR;
      =     #OK;	// CFB execution OK
      O     #STAT;	// WARNING/ERROR
      O     #ERROR;	// ERROR
      R     #OK;	// CFB execution not OK
      S     #NOT_OK;
END_FUNCTION

FUNCTION "EXAMPLE_URCV" : VOID	// FC 104
VERSION : 0.0
BEGIN
NETWORK
TITLE =
      A     "en_r_urcv_user";	//*If "en_r" 0->1,
      FP    "data_urcv".edge;
      JCN   m1;
      L     0;	//*reset
      T     "data_urcv".saved_status;	//*saved STATUS 
m1:   NOP   0;
      BLD   9;
      =     L 4.0;
      CDB;
      OPN   DI 9;
      TAR2  LD 0;
      A     "en_r_urcv_user";
      =     DIX 0.0;
      OPN   DI 101;
      L     DIW 2;
      OPN   DI 9;
      T     DIW 2;
      OPN   DI 101;	//*If STATUS is not "0",
      L     DID 4;	//*
      OPN   DI 9;	//*
      T     DID 4;
      L     W#16#1002;	//*
      T     DIW 12;	//*set "not_ok"
      L     30;	//*and save STATUS
      T     DIW 14;
      L     101;
//                                      //Add troubleshooting routine h             
      T     DIW 16;
      L     P#DBX 10.0;
      T     DID 18;
      L     W#16#1002;
      T     DIW 22;
      L     30;
      T     DIW 24;
      L     101;
      T     DIW 26;
      L     P#DBX 110.0;
      T     DID 28;
      L     W#16#1002;
      T     DIW 32;
      L     30;
      T     DIW 34;
      L     101;
      T     DIW 36;
      L     P#DBX 210.0;
      T     DID 38;
      L     W#16#1002;
      T     DIW 42;
      L     30;
      T     DIW 44;
      L     101;
      T     DIW 46;
      L     P#DBX 310.0;
      T     DID 48;
      LAR2  P#DBX 0.0;
      UC    "URCV";
      LAR2  LD 0;
      A     DIX 8.0;
      OPN   DI 101;
      =     DIX 0.1;
      OPN   DI 9;
      A     DIX 8.1;
      OPN   DI 101;
      =     DIX 0.2;
      OPN   DI 9;
      L     DIW 10;
      OPN   DI 101;
      T     DIW 8;
      OPN   DI 9;
      CDB;
      BLD   10;
      L     0;
      L     "data_urcv".status;
      <>I;
      JCN   mark;
      SET;
      =     "data_urcv".not_ok;
      T     "data_urcv".saved_status;
mark: NOP   0;
      A     "data_urcv".not_ok;
END_FUNCTION

FUNCTION "EXAMPLE_BRCV" : VOID	// FC 106
VERSION : 0.0
BEGIN
NETWORK
TITLE =
      A     "en_r_brcv_user";	//*If "en_r" 0->1,
      FP    "data_brcv".edge;
      JCN   m1;
      L     0;	//*reset
      T     "data_brcv".saved_status;	//*saved STATUS 
m1:   NOP   0;
      BLD   9;
      =     L 4.0;
      CDB;
      OPN   DI 13;
      TAR2  LD 0;
      A     "en_r_brcv_user";
      =     DIX 0.0;
      OPN   DI 103;
      L     DIW 2;
      OPN   DI 13;	//*If STATUS is not "0",
      T     DIW 2;	//*
      OPN   DI 103;	//*
      L     DID 4;
      OPN   DI 13;	//*
      T     DID 4;	//*set "not_ok"
      L     W#16#1002;	//*and save STATUS
      T     DIW 12;
      L     500;
//                                      //Add troubleshooting routine h             
      T     DIW 14;
      L     103;
      T     DIW 16;
      L     P#DBX 12.0;
      T     DID 18;
      OPN   DI 103;
      L     DIW 10;
      OPN   DI 13;
      T     DIW 22;
      LAR2  P#DBX 0.0;
      UC    "BRCV";
      LAR2  LD 0;
      A     DIX 8.0;
      OPN   DI 103;
      =     DIX 0.1;
      OPN   DI 13;
      A     DIX 8.1;
      OPN   DI 103;
      =     DIX 0.2;
      OPN   DI 13;
      L     DIW 10;
      OPN   DI 103;
      T     DIW 8;
      OPN   DI 13;
      L     DIW 22;
      OPN   DI 103;
      T     DIW 10;
      OPN   DI 13;
      CDB;
      BLD   10;
      L     0;
      L     "data_brcv".status;
      <>I;
      JCN   mark;
      SET;
      =     "data_brcv".not_ok;
      T     "data_brcv".saved_status;
mark: NOP   0;
      A     "data_brcv".not_ok;
END_FUNCTION

FUNCTION "EXAMPLE_PRESET_SFBs_2" : VOID	// FC 112
TITLE = *****              INITIALIZING CFBs           *****
VERSION : 2.0
BEGIN
NETWORK
TITLE =  INITIALIZING URCV 
      CLR;
      =     "en_r_urcv_user";
      L     W#16#1;	// connection_id
      T     "data_urcv".id;
      L     DW#16#80009;	// 
      T     "data_urcv".r_id;
      L     W#16#0;
      T     "data_urcv".saved_status;
NETWORK
TITLE =  INITIALIZING BRCV 
      CLR;
      =     "en_r_brcv_user";
      L     W#16#1;	// connection_id
      T     "data_brcv".id;
      L     DW#16#C000D;
      T     "data_brcv".r_id;
      L     W#16#0;
      T     "data_brcv".saved_status;
NETWORK
TITLE =  Presetting the send values for GET 
// DB107 Byte 0-399
      L     W#16#101;
      T     "data_get_source".fill_1;
      CALL  "FILL" (
           BVAL                     := "data_get_source".fill_1,
           RET_VAL                  := "data_get_source".ret_val,
           BLK                      := "data_get_source".source_1);
//  
      L     W#16#202;
      T     "data_get_source".fill_2;
      CALL  "FILL" (
           BVAL                     := "data_get_source".fill_2,
           RET_VAL                  := "data_get_source".ret_val,
           BLK                      := "data_get_source".source_2);
//  
      L     W#16#303;
      T     "data_get_source".fill_3;
      CALL  "FILL" (
           BVAL                     := "data_get_source".fill_3,
           RET_VAL                  := "data_get_source".ret_val,
           BLK                      := "data_get_source".source_3);
//  
      L     W#16#404;
      T     "data_get_source".fill_4;
      CALL  "FILL" (
           BVAL                     := "data_get_source".fill_4,
           RET_VAL                  := "data_get_source".ret_val,
           BLK                      := "data_get_source".source_4);
//  
NETWORK
TITLE =  Presetting destination area for PUT
      L     W#16#0;
      T     "data_put_destination".fill;
      CALL  "FILL" (
           BVAL                     := "data_put_destination".fill,
           RET_VAL                  := "data_put_destination".ret_val,
           BLK                      := "data_put_destination".dest_1);
      CALL  "FILL" (
           BVAL                     := "data_put_destination".fill,
           RET_VAL                  := "data_put_destination".ret_val,
           BLK                      := "data_put_destination".dest_2);
      CALL  "FILL" (
           BVAL                     := "data_put_destination".fill,
           RET_VAL                  := "data_put_destination".ret_val,
           BLK                      := "data_put_destination".dest_3);
      CALL  "FILL" (
           BVAL                     := "data_put_destination".fill,
           RET_VAL                  := "data_put_destination".ret_val,
           BLK                      := "data_put_destination".dest_4);
NETWORK
TITLE =  Presetting destination area for URCV
      L     W#16#0;
      T     "data_urcv".fill;
      CALL  "FILL" (
           BVAL                     := "data_urcv".fill,
           RET_VAL                  := "data_urcv".ret_val,
           BLK                      := "data_urcv".rcv_data_1);
      CALL  "FILL" (
           BVAL                     := "data_urcv".fill,
           RET_VAL                  := "data_urcv".ret_val,
           BLK                      := "data_urcv".rcv_data_2);
      CALL  "FILL" (
           BVAL                     := "data_urcv".fill,
           RET_VAL                  := "data_urcv".ret_val,
           BLK                      := "data_urcv".rcv_data_3);
      CALL  "FILL" (
           BVAL                     := "data_urcv".fill,
           RET_VAL                  := "data_urcv".ret_val,
           BLK                      := "data_urcv".rcv_data_4);
NETWORK
TITLE =  Presetting destination area for BRCV
      L     W#16#0;
      T     "data_brcv".fill;
      CALL  "FILL" (
           BVAL                     := "data_brcv".fill,
           RET_VAL                  := "data_brcv".ret_val,
           BLK                      := "data_brcv".rcv_data_1);
NETWORK
TITLE = BLOCK_END
END_FUNCTION

DATA_BLOCK "IDB_URCV"	// DB 9
VERSION : 0.0
"URCV"
BEGIN
END_DATA_BLOCK

DATA_BLOCK "IDB_BRCV"	// DB 13
VERSION : 0.0
"BRCV"
BEGIN
END_DATA_BLOCK

DATA_BLOCK "data_urcv"	// DB 101
VERSION : 2.0
  STRUCT
   en_r : BOOL ;	//Can be used if needed
   ndr : BOOL ;
   error : BOOL ;
   busy : BOOL ;	//Can be used if needed
   ok : BOOL ;
   not_ok : BOOL ;
   id : WORD ;
   r_id : DWORD ;
   status : WORD ;
   rcv_data_1 : ARRAY  [1 .. 30 ] OF BYTE ;
   erw_rcv_data_1 : ARRAY  [1 .. 70 ] OF BYTE ;
   rcv_data_2 : ARRAY  [1 .. 30 ] OF BYTE ;
   erw_rcv_data_2 : ARRAY  [1 .. 70 ] OF BYTE ;
   rcv_data_3 : ARRAY  [1 .. 30 ] OF BYTE ;
   erw_rcv_data_3 : ARRAY  [1 .. 70 ] OF BYTE ;
   rcv_data_4 : ARRAY  [1 .. 30 ] OF BYTE ;
   erw_rcv_data_4 : ARRAY  [1 .. 70 ] OF BYTE ;
   fill : WORD ;
   ret_val : INT ;
   saved_status : WORD ;
   edge : BOOL ;
  END_STRUCT ;	
BEGIN
   en_r := TRUE;
   id := W#16#1;
   r_id := DW#16#80009;
   rcv_data_1[1] := B#16#1;
   rcv_data_1[2] := B#16#1;
   rcv_data_1[3] := B#16#1;
   rcv_data_1[4] := B#16#1;
   rcv_data_1[5] := B#16#1;
   rcv_data_1[6] := B#16#1;
   rcv_data_1[7] := B#16#1;
   rcv_data_1[8] := B#16#1;
   rcv_data_1[9] := B#16#1;
   rcv_data_1[10] := B#16#1;
   rcv_data_2[1] := B#16#2;
   rcv_data_2[2] := B#16#2;
   rcv_data_2[3] := B#16#2;
   rcv_data_2[4] := B#16#2;
   rcv_data_2[5] := B#16#2;
   rcv_data_2[6] := B#16#2;
   rcv_data_2[7] := B#16#2;
   rcv_data_2[8] := B#16#2;
   rcv_data_2[9] := B#16#2;
   rcv_data_2[10] := B#16#2;
   rcv_data_2[11] := B#16#2;
   rcv_data_2[12] := B#16#2;
   rcv_data_2[13] := B#16#2;
   rcv_data_2[14] := B#16#2;
   rcv_data_2[15] := B#16#2;
   rcv_data_2[16] := B#16#2;
   rcv_data_2[17] := B#16#2;
   rcv_data_2[18] := B#16#2;
   rcv_data_2[19] := B#16#2;
   rcv_data_2[20] := B#16#2;
   rcv_data_2[21] := B#16#2;
   rcv_data_2[22] := B#16#2;
   rcv_data_2[23] := B#16#2;
   rcv_data_2[24] := B#16#2;
   rcv_data_2[25] := B#16#2;
   rcv_data_2[26] := B#16#2;
   rcv_data_2[27] := B#16#2;
   rcv_data_2[28] := B#16#2;
   rcv_data_2[29] := B#16#2;
   rcv_data_2[30] := B#16#2;
   rcv_data_3[1] := B#16#3;
   rcv_data_3[2] := B#16#3;
   rcv_data_3[3] := B#16#3;
   rcv_data_3[4] := B#16#3;
   rcv_data_3[5] := B#16#3;
   rcv_data_3[6] := B#16#3;
   rcv_data_3[7] := B#16#3;
   rcv_data_3[8] := B#16#3;
   rcv_data_3[9] := B#16#3;
   rcv_data_3[10] := B#16#3;
   rcv_data_3[11] := B#16#3;
   rcv_data_3[12] := B#16#3;
   rcv_data_3[13] := B#16#3;
   rcv_data_3[14] := B#16#3;
   rcv_data_3[15] := B#16#3;
   rcv_data_3[16] := B#16#3;
   rcv_data_3[17] := B#16#3;
   rcv_data_3[18] := B#16#3;
   rcv_data_3[19] := B#16#3;
   rcv_data_3[20] := B#16#3;
   rcv_data_3[21] := B#16#3;
   rcv_data_3[22] := B#16#3;
   rcv_data_3[23] := B#16#3;
   rcv_data_3[24] := B#16#3;
   rcv_data_3[25] := B#16#3;
   rcv_data_3[26] := B#16#3;
   rcv_data_3[27] := B#16#3;
   rcv_data_3[28] := B#16#3;
   rcv_data_3[29] := B#16#3;
   rcv_data_3[30] := B#16#3;
   rcv_data_4[1] := B#16#4;
   rcv_data_4[2] := B#16#4;
   rcv_data_4[3] := B#16#4;
   rcv_data_4[4] := B#16#4;
   rcv_data_4[5] := B#16#4;
   rcv_data_4[6] := B#16#4;
   rcv_data_4[7] := B#16#4;
   rcv_data_4[8] := B#16#4;
   rcv_data_4[9] := B#16#4;
   rcv_data_4[10] := B#16#4;
   rcv_data_4[11] := B#16#4;
   rcv_data_4[12] := B#16#4;
   rcv_data_4[13] := B#16#4;
   rcv_data_4[14] := B#16#4;
   rcv_data_4[15] := B#16#4;
   rcv_data_4[16] := B#16#4;
   rcv_data_4[17] := B#16#4;
   rcv_data_4[18] := B#16#4;
   rcv_data_4[19] := B#16#4;
   rcv_data_4[20] := B#16#4;
   rcv_data_4[21] := B#16#4;
   rcv_data_4[22] := B#16#4;
   rcv_data_4[23] := B#16#4;
   rcv_data_4[24] := B#16#4;
   rcv_data_4[25] := B#16#4;
   rcv_data_4[26] := B#16#4;
   rcv_data_4[27] := B#16#4;
   rcv_data_4[28] := B#16#4;
   rcv_data_4[29] := B#16#4;
   rcv_data_4[30] := B#16#4;
END_DATA_BLOCK

DATA_BLOCK "data_brcv"	// DB 103
VERSION : 0.0
  STRUCT
   en_r : BOOL ;	//Can be used if needed
   ndr : BOOL ;
   error : BOOL ;
   busy : BOOL ;	//Can be used if needed
   ok : BOOL ;
   not_ok : BOOL ;
   id : WORD ;
   r_id : DWORD ;
   status : WORD ;
   len : WORD ;
   rcv_data_1 : ARRAY  [1 .. 500 ] OF BYTE ;
   erw_rcv_data_1 : ARRAY  [1 .. 500 ] OF BYTE ;
   fill : WORD ;
   ret_val : INT ;
   saved_status : WORD ;
   edge : BOOL ;
  END_STRUCT ;	
BEGIN
END_DATA_BLOCK

DATA_BLOCK "data_get_source"	// DB 107
VERSION : 0.1
  STRUCT
   source_1 : ARRAY  [1 .. 100 ] OF BYTE ;
   source_2 : ARRAY  [1 .. 100 ] OF BYTE ;
   source_3 : ARRAY  [1 .. 100 ] OF BYTE ;
   source_4 : ARRAY  [1 .. 100 ] OF BYTE ;
   fill_1 : WORD ;
   fill_2 : WORD ;
   fill_3 : WORD ;
   fill_4 : WORD ;
   ret_val : INT ;
  END_STRUCT ;	
BEGIN
END_DATA_BLOCK

DATA_BLOCK "data_put_destination"	// DB 108
VERSION : 0.1
  STRUCT
   dest_1 : ARRAY  [1 .. 100 ] OF BYTE ;
   dest_2 : ARRAY  [1 .. 100 ] OF BYTE ;
   dest_3 : ARRAY  [1 .. 100 ] OF BYTE ;
   dest_4 : ARRAY  [1 .. 100 ] OF BYTE ;
   fill : WORD ;
   ret_val : INT ;
  END_STRUCT ;	
BEGIN
END_DATA_BLOCK

ORGANIZATION_BLOCK "CYC_INT5"	// OB 35
TITLE = "100 ms Cycle"
VERSION : 1.0
VAR_TEMP
  OB35_EV_CLASS : BYTE ;
  OB35_STRT_INF : BYTE ;
  OB35_PRIORITY : BYTE ;
  OB35_OB_NUMBR : BYTE ;
  OB35_RESERVED_1 : BYTE ;
  OB35_RESERVED_2 : BYTE ;
  OB35_PHASE_OFFSET : WORD ;
  OB35_RESERVED_3 : INT ;
  OB35_EXC_FREQ : INT ;
  OB35_DATE_TIME : DATE_AND_TIME ;
END_VAR
BEGIN
NETWORK
TITLE = CALL URCV
      CALL  "EXAMPLE_URCV";
NETWORK
TITLE = CALL BRCV
      CALL  "EXAMPLE_BRCV";
END_ORGANIZATION_BLOCK

ORGANIZATION_BLOCK "COMPLETE RESTART"	// OB 100
TITLE = "Complete Restart"
VERSION : 1.0
VAR_TEMP
  OB100_EV_CLASS : BYTE ;
  OB100_STRTUP : BYTE ;
  OB100_PRIORITY : BYTE ;
  OB100_OB_NUMBR : BYTE ;
  OB100_RESERVED_1 : BYTE ;
  OB100_RESERVED_2 : BYTE ;
  OB100_STOP : WORD ;
  OB100_STRT_INFO : DWORD ;
  OB100_DATE_TIME : DATE_AND_TIME ;
END_VAR
BEGIN
NETWORK
TITLE = ***** INITIALIZING RECIEVE SFBs                ******
      CALL  "EXAMPLE_PRESET_SFBs_2";
END_ORGANIZATION_BLOCK
